// TIA Portal project "Task2" (V16)

(* hardware
DEVICE "S7-1200 station_1"  S7-1200 Station
   slot 0: "Rack_0"  S7-1200 Rack  Rack  V1.0
   slot 1: "PLC_LEFT"  CPU 1214C AC/DC/Rly  6ES7 214-1BG40-0XB0  V4.1
   slot 2: "DI 8/DQ 8x24VDC_1"  6ES7 223-1BH32-0XB0  V2.0
DEVICE "S7-1200 station_2"  S7-1200 Station
   slot 0: "Rack_0"  S7-1200 Rack  Rack  V1.0
   slot 1: "PLC_MIDDLE"  CPU 1214C AC/DC/Rly  6ES7 214-1BG40-0XB0  V4.4
   slot 2: "DI 8/DQ 8x24VDC_1"  6ES7 223-1BH32-0XB0  V2.0
   slot 3: "AI 4x13BIT/AQ 2x14BIT_1"  6ES7 234-4HE32-0XB0  V2.0
DEVICE "S7-1200 station_3"  S7-1200 Station
   slot 0: "Rack_0"  S7-1200 Rack  Rack  V1.0
   slot 1: "PLC_RIGHT"  CPU 1214C AC/DC/Rly  6ES7 214-1BG40-0XB0  V4.1
   slot 2: "DI 8/DQ 8x24VDC_1"  6ES7 223-1BH32-0XB0  V2.0
   slot 3: "AI 4x13BIT/AQ 2x14BIT_1"  6ES7 234-4HE32-0XB0  V2.0
*)

// ===== PLC "PLC_LEFT"  CPU 1214C AC/DC/Rly =====

VAR_GLOBAL   // PLC tag table "Default tag table"
   "Tag_1" AT %M8.0 : Bool;
   "System_Byte" AT %MB1 : Byte;
   "FirstScan" AT %M1.0 : Bool;
   "DiagStatusUpdate" AT %M1.1 : Bool;
   "AlwaysTRUE" AT %M1.2 : Bool;
   "AlwaysFALSE" AT %M1.3 : Bool;
   "Clock_Byte" AT %MB0 : Byte;
   "Clock_10Hz" AT %M0.0 : Bool;
   "Clock_5Hz" AT %M0.1 : Bool;
   "Clock_2.5Hz" AT %M0.2 : Bool;
   "Clock_2Hz" AT %M0.3 : Bool;
   "Clock_1.25Hz" AT %M0.4 : Bool;
   "Clock_1Hz" AT %M0.5 : Bool;
   "Clock_0.625Hz" AT %M0.6 : Bool;
   "Clock_0.5Hz" AT %M0.7 : Bool;
END_VAR

VAR_GLOBAL   // PLC tag table "INPUT"
   "processing_input_5_carousel_init" AT %I8.5 : Bool;
   "processing_input_6_hole_detected" AT %I8.6 : Bool;
   "processing_input_1_workpiece_detected" AT %I8.1 : Bool;
   "processing_input_7_workpiece_not_black" AT %I8.7 : Bool;
   "processing_input_2_workpiece_silver" AT %I8.2 : Bool;
END_VAR

VAR_GLOBAL   // PLC tag table "OUTPUT"
   "processing_output_0_drill" AT %Q8.0 : Bool;
   "processing_output_1_rotate_carousel" AT %Q8.1 : Bool;
   "processing_output_2_drill_down" AT %Q8.2 : Bool;
   "processing_output_3_drill_up" AT %Q8.3 : Bool;
   "processing_output_4_fix_workpiece" AT %Q8.4 : Bool;
   "processing_output_5_detect_hole" AT %Q8.5 : Bool;
END_VAR

ORGANIZATION_BLOCK "Main"   // OB1, LAD, ProgramCycle
TITLE = "Main Program Sweep (Cycle)"
{ S7_Optimized_Access := 'TRUE' }
VERSION : 0.1
   VAR_INPUT
      Initial_Call : Bool;   // Initial call of this OB
      Remanence : Bool;   // =True, if remanent data are available
   END_VAR
BEGIN

REGION Network 1
   // PUT 4 tags to middle PLC
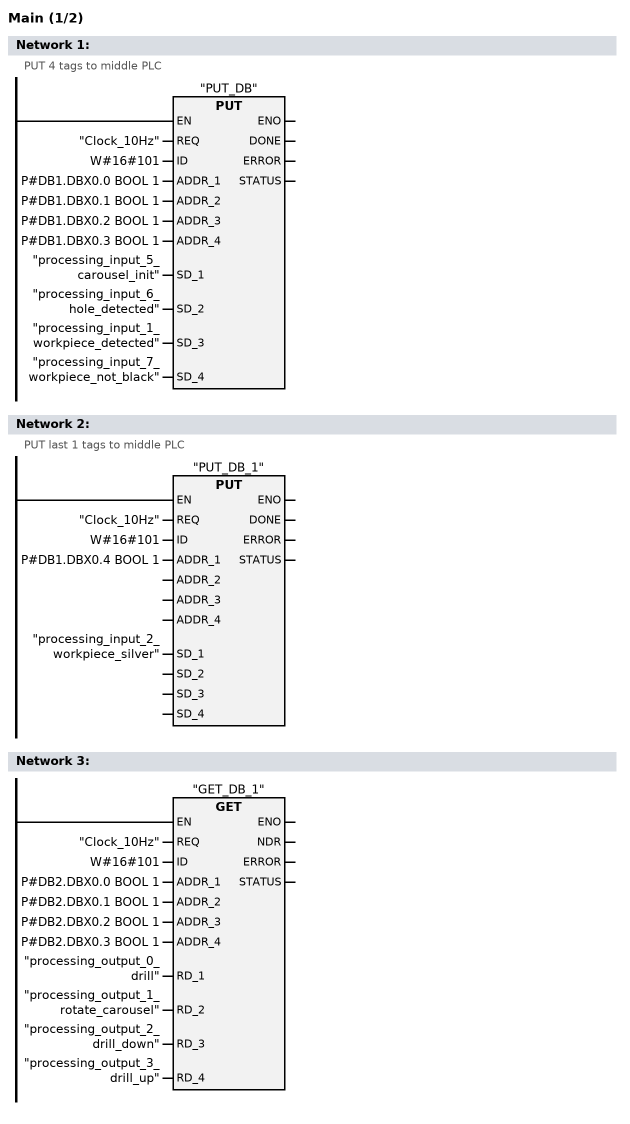
   "PUT_DB"(REQ := "Clock_10Hz",   // PUT
            ID := W#16#101,
            ADDR_1 := P#DB1.DBX0.0 BOOL 1,
            ADDR_2 := P#DB1.DBX0.1 BOOL 1,
            ADDR_3 := P#DB1.DBX0.2 BOOL 1,
            ADDR_4 := P#DB1.DBX0.3 BOOL 1,
            SD_1 := "processing_input_5_carousel_init",
            SD_2 := "processing_input_6_hole_detected",
            SD_3 := "processing_input_1_workpiece_detected",
            SD_4 := "processing_input_7_workpiece_not_black");
END_REGION

REGION Network 2
   // PUT last 1 tags to middle PLC
   "PUT_DB_1"(REQ := "Clock_10Hz",   // PUT
              ID := W#16#101,
              ADDR_1 := P#DB1.DBX0.4 BOOL 1,
              SD_1 := "processing_input_2_workpiece_silver");
END_REGION

REGION Network 3
   "GET_DB_1"(REQ := "Clock_10Hz",   // GET
              ID := W#16#101,
              ADDR_1 := P#DB2.DBX0.0 BOOL 1,
              ADDR_2 := P#DB2.DBX0.1 BOOL 1,
              ADDR_3 := P#DB2.DBX0.2 BOOL 1,
              ADDR_4 := P#DB2.DBX0.3 BOOL 1,
              RD_1 := "processing_output_0_drill",
              RD_2 := "processing_output_1_rotate_carousel",
              RD_3 := "processing_output_2_drill_down",
              RD_4 := "processing_output_3_drill_up");
END_REGION

REGION Network 4
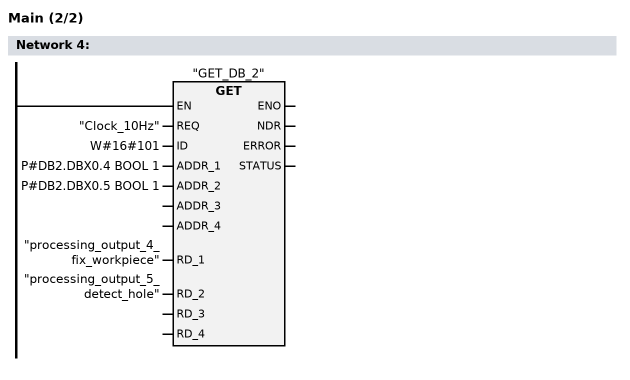
   "GET_DB_2"(REQ := "Clock_10Hz",   // GET
              ID := W#16#101,
              ADDR_1 := P#DB2.DBX0.4 BOOL 1,
              ADDR_2 := P#DB2.DBX0.5 BOOL 1,
              RD_1 := "processing_output_4_fix_workpiece",
              RD_2 := "processing_output_5_detect_hole");
END_REGION
END_ORGANIZATION_BLOCK

// ===== PLC "PLC_MIDDLE"  CPU 1214C AC/DC/Rly =====

VAR_GLOBAL   // PLC tag table "Default tag table"
   "packing_input_7_pack_turned_on" AT %I0.7 : Bool;
   "packing_output_4_push_box" AT %Q0.4 : Bool;
   "packing_output_5_fix_box_upper_side" AT %Q0.5 : Bool;
   "packing_output_6_fix_box_tongue" AT %Q0.6 : Bool;
   "packing_output_7_pack_box" AT %Q0.7 : Bool;
   "Tag_1" AT %M8.0 : Bool;
   "Tag_2" AT %M8.1 : Bool;
   "Tag_3" AT %M8.2 : Bool;
END_VAR

VAR_GLOBAL   // PLC tag table "INPUT"
   "handling_input_3_gripper_at_right" AT %I8.3 : Bool;
   "handling_input_2_gripper_at_start" AT %I8.2 : Bool;
   "handling_input_1_gripper_at_packing_station" AT %I8.1 : Bool;
   "handling_input_0_workpiece_pushed" AT %I8.0 : Bool;
   "handling_input_4_gripper_down_pack_lvl" AT %I8.4 : Bool;
END_VAR

VAR_GLOBAL   // PLC tag table "OUTPUT"
   "handling_output_0_to_green" AT %Q8.0 : Bool;
   "handling_output_7_push_workpiece" AT %Q8.7 : Bool;
   "handling_output_6_gripper_to_open" AT %Q8.6 : Bool;
   "handling_output_5_gripper_to_down" AT %Q8.5 : Bool;
   "handling_output_4_gripper_to_left" AT %Q8.4 : Bool;
   "handling_output_3_gripper_to_right" AT %Q8.3 : Bool;
   "handling_output_2_to_red" AT %Q8.2 : Bool;
   "handling_output_1_to_yellow" AT %Q8.1 : Bool;
END_VAR

DATA_BLOCK "DB_FROM_LEFT"   // DB1
{ S7_Optimized_Access := 'FALSE' }
VERSION : 0.1
   VAR
      processing_input_5_carousel_init : Bool;
      processing_input_6_hole_detected : Bool;
      processing_input_1_workpiece_detected : Bool;
      processing_input_7_workpiece_not_black : Bool;
      processing_input_2_workpiece_silver : Bool;
   END_VAR
BEGIN
END_DATA_BLOCK

DATA_BLOCK "DB_TO_LEFT"   // DB2
{ S7_Optimized_Access := 'FALSE' }
VERSION : 0.1
   VAR
      processing_output_0_drill : Bool;
      processing_output_1_rotate_carousel : Bool;
      processing_output_2_drill_down : Bool;
      processing_output_3_drill_up : Bool;
      processing_output_4_fix_workpiece : Bool;
      processing_output_5_detect_hole : Bool;
   END_VAR
BEGIN
END_DATA_BLOCK

DATA_BLOCK "DB_FROM_RIGHT"   // DB3
{ S7_Optimized_Access := 'FALSE' }
VERSION : 0.1
   VAR
      sorting_input_3_box_on_conveyor : Bool;
      sorting_input_4_box_is_down : Bool;
   END_VAR
BEGIN
END_DATA_BLOCK

DATA_BLOCK "DB_TO_RIGHT"   // DB4
{ S7_Optimized_Access := 'FALSE' }
VERSION : 0.1
   VAR
      sorting_output_0_move_conveyor_right : Bool;
      sorting_output_1_move_conveyor_left : Bool;
      sorting_output_2_push_silver_workpiece : Bool;
      sorting_output_3_push_red_workpiece : Bool;
   END_VAR
BEGIN
END_DATA_BLOCK

DATA_BLOCK "ADDITIONAL_VARIABLES"   // DB5
{ S7_Optimized_Access := 'FALSE' }
VERSION : 0.1
   VAR
      Red : Bool;
      Black : Bool;
      Silvery : Bool;
      Stop : Bool;
      Reset : Bool;
      Start : Bool;
      "Step" : Int;
   END_VAR
BEGIN
END_DATA_BLOCK

DATA_BLOCK "main_db"   // DB6
{ S7_Optimized_Access := 'TRUE' }
VERSION : 0.1
BEGIN
END_DATA_BLOCK

ORGANIZATION_BLOCK "Main"   // OB1, SCL, ProgramCycle
TITLE = "Main Program Sweep (Cycle)"
{ S7_Optimized_Access := 'TRUE' }
VERSION : 0.1
   VAR_INPUT
      Initial_Call : Bool;   // Initial call of this OB
      Remanence : Bool;   // =True, if remanent data are available
   END_VAR
BEGIN

       // Кнопка стоп
   IF "ADDITIONAL_VARIABLES".Stop THEN

   END_IF;
       // Кнопка старт
   IF "ADDITIONAL_VARIABLES".Start THEN

   END_IF;
END_ORGANIZATION_BLOCK

// ===== PLC "PLC_RIGHT"  CPU 1214C AC/DC/Rly =====

VAR_GLOBAL   // PLC tag table "Default tag table"
   "Clock_10Hz" AT %M0.0 : Bool;
   "System_Byte" AT %MB1 : Byte;
   "FirstScan" AT %M1.0 : Bool;
   "DiagStatusUpdate" AT %M1.1 : Bool;
   "AlwaysTRUE" AT %M1.2 : Bool;
   "AlwaysFALSE" AT %M1.3 : Bool;
   "Clock_Byte" AT %MB0 : Byte;
   "Clock_5Hz" AT %M0.1 : Bool;
   "Clock_2.5Hz" AT %M0.2 : Bool;
   "Clock_2Hz" AT %M0.3 : Bool;
   "Clock_1.25Hz" AT %M0.4 : Bool;
   "Clock_1Hz" AT %M0.5 : Bool;
   "Clock_0.625Hz" AT %M0.6 : Bool;
   "Clock_0.5Hz" AT %M0.7 : Bool;
END_VAR

VAR_GLOBAL   // PLC tag table "INPUT"
   "sorting_input_4_box_is_down" AT %I8.4 : Bool;
   "sorting_input_3_box_on_conveyor" AT %I8.3 : Bool;
END_VAR

VAR_GLOBAL   // PLC tag table "OUTPUT"
   "sorting_output_0_move_conveyor_right" AT %Q8.0 : Bool;
   "sorting_output_1_move_conveyor_left" AT %Q8.1 : Bool;
   "sorting_output_2_push_silver_workpiece" AT %Q8.3 : Bool;
   "sorting_output_3_push_red_workpiece" AT %Q8.2 : Bool;
END_VAR

ORGANIZATION_BLOCK "Main"   // OB1, LAD, ProgramCycle
TITLE = "Main Program Sweep (Cycle)"
{ S7_Optimized_Access := 'TRUE' }
VERSION : 0.1
   VAR_INPUT
      Initial_Call : Bool;   // Initial call of this OB
      Remanence : Bool;   // =True, if remanent data are available
   END_VAR
BEGIN

REGION Network 1
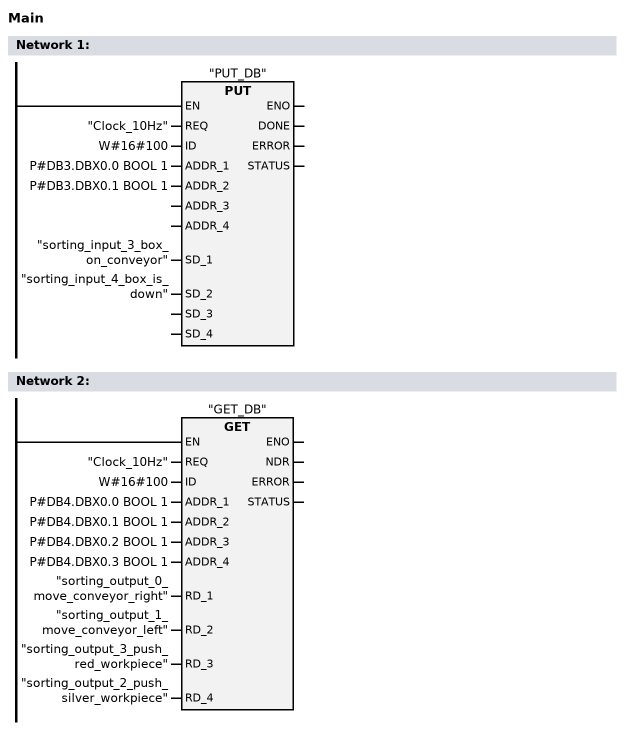
   "PUT_DB"(REQ := "Clock_10Hz",   // PUT
            ID := W#16#100,
            ADDR_1 := P#DB3.DBX0.0 BOOL 1,
            ADDR_2 := P#DB3.DBX0.1 BOOL 1,
            SD_1 := "sorting_input_3_box_on_conveyor",
            SD_2 := "sorting_input_4_box_is_down");
END_REGION

REGION Network 2
   "GET_DB"(REQ := "Clock_10Hz",   // GET
            ID := W#16#100,
            ADDR_1 := P#DB4.DBX0.0 BOOL 1,
            ADDR_2 := P#DB4.DBX0.1 BOOL 1,
            ADDR_3 := P#DB4.DBX0.2 BOOL 1,
            ADDR_4 := P#DB4.DBX0.3 BOOL 1,
            RD_1 := "sorting_output_0_move_conveyor_right",
            RD_2 := "sorting_output_1_move_conveyor_left",
            RD_3 := "sorting_output_3_push_red_workpiece",
            RD_4 := "sorting_output_2_push_silver_workpiece");
END_REGION
END_ORGANIZATION_BLOCK